// TIA Portal V15.1 export
// export: Created 2024-05-17T05:38:41.5679982Z, ExportSetting WithDefaults, DisplayName Totally Integrated Automation Portal, DisplayVersion V15.1 Update 5, DisplayName TIA Portal Openness, DisplayVersion V15.1 Update 5, DisplayName SINAMICS Startdrive Advanced, DisplayVersion V15.1, DisplayName G130, G150, S120, S150, SINAMICS MV, S210, DisplayVersion V15.1, DisplayName G110M, G120, G120C, G120D, G120P, DisplayVersion V15.1, DisplayName STEP 7 Professional, DisplayVersion V15.1 Update 5, DisplayName STEP 7 Safety, DisplayVersion V15.1, DisplayName WinCC Professional, DisplayVersion V15.1 Update 5, DisplayName SIMATIC Visualization Architect, DisplayVersion V15.1
FUNCTION "LGBLineConvBrake-MDXPN-DFS22B-Config" : Void   // FC6713, FBD
TITLE = LCrossConv2W2S-G120PN-Config / LGBLineConvBrake-MDXPN-DFS22B-Config
{ S7_Optimized_Access := 'FALSE' }
AUTHOR : VCC
FAMILY : Config
NAME : Bit2Word
VERSION : 0.1
// =============================================================================
// Handles the LCross2W2SG120PN Config
// =============================================================================
// stored: AutoNumber false, IsIECCheckEnabled false, SetENOAutomatically False, UDAEnableTagReadback false
   VAR_INPUT
      C_DetBeltTensionUsed : Bool;   // Input 0 / Config / Lowspeed stop detection Set used
      C_DetMinGapLeftUsed : Bool;   // Input 0 / Config / Lowspeed stop detection Set used
      C_DetMinGapRightUsed : Bool;   // Input 0 / Config / Lowspeed stop detection Set used
      C_BothDetMinGapIsAlarmB : Bool;   // Config
      C_OneDetMinGapIsAlarmC : Bool;   // Config
      C_InitDirectionMotPower : Bool;   // Input 7 / Config
      C_InitDirectionMotBrake : Bool;   // Input 7 / Config
      C_SafetySwNcMotPower : Bool;   // Input 15 / Config
      C_SafetySwUsedMotPower : Bool;   // Input 16 / Config
      C_SafetySwNcMotBrake : Bool;   // Input 15 / Config
      C_SafetySwUsedMotBrake : Bool;   // Input 16 / Config
      C_MotorProtectionNc : Bool;   // Motorprotection NC / Config
      C_MotorProtectionUsed : Bool;   // Motorprotection NC / Config
      C_BrakeProtectionNc : Bool;   // Config
      C_BrakeProtectionUsed : Bool;   // Config
      C_MotionStopUsed : Bool;   // Config
      C_EnableAlarmHW : Bool;   // Enable Alarm hardware (e.g. safetyswitch, motorprotector, detections) / Enable Alarm hardware (e.g. Safetyswitch, Motorprotector, detections) / Config
      C_EnableAlarmTransfer : Bool;   // Enable Alarm transfer (e.g. Transfer in , transfer out) / Config
      C_DetSaturationDelay : Time;   // Config
      C_RampMotBrake : Time;   // Config
      C_ReferenceDriveCurrentMotBrake : Real;   // Config
      C_ReferenceMotorCurrentMotBrake : Real;   // Config
      C_ReferenceMotorRPMMotBrake : Real;   // Config
      C_RatioGearboxMotBrake : Real;   // Config
      C_DiameterMotBrake : Real;   // Config
      C_AccelerationMotBrake : Real;   // Config
      C_RampMotPower : Time;   // Config
      C_ReferenceDriveCurrentMotPower : Real;   // Config
      C_ReferenceMotorCurrentMotPower : Real;   // Config
      C_ReferenceMotorRPMMotPower : Real;   // Config
      C_RatioGearboxMotPower : Real;   // Config
      C_DiameterMotPower : Real;   // Config
      C_AccelerationMotPower : Real;   // Config
      C_TrfMaxTime : DInt;   // Max allowed transfertime (millisec) / Config
      C_AllowedResetDirection : Bool;   // Config
      C_MaxTimeResetDirection : DInt;   // Config
      C_AllowedEcoMode : Bool;   // Config
      C_TimeEcoMode : Time;   // Config
      C_HWSubInputMotPower : HW_SUBMODULE;   // I/O / Config
      C_HWSubOutputMotPower : HW_SUBMODULE;   // I/O / Config
      C_HWSubInputMotBrake : HW_SUBMODULE;   // I/O / Config
      C_HWSubOutputMotBrake : HW_SUBMODULE;   // I/O / Config
   END_VAR
   VAR_IN_OUT
      IO_Config : "LineConvBrake-MDXPNConfig";   // Config
   END_VAR
BEGIN

REGION Network 1: **** 1 - Inputs **** Move Config
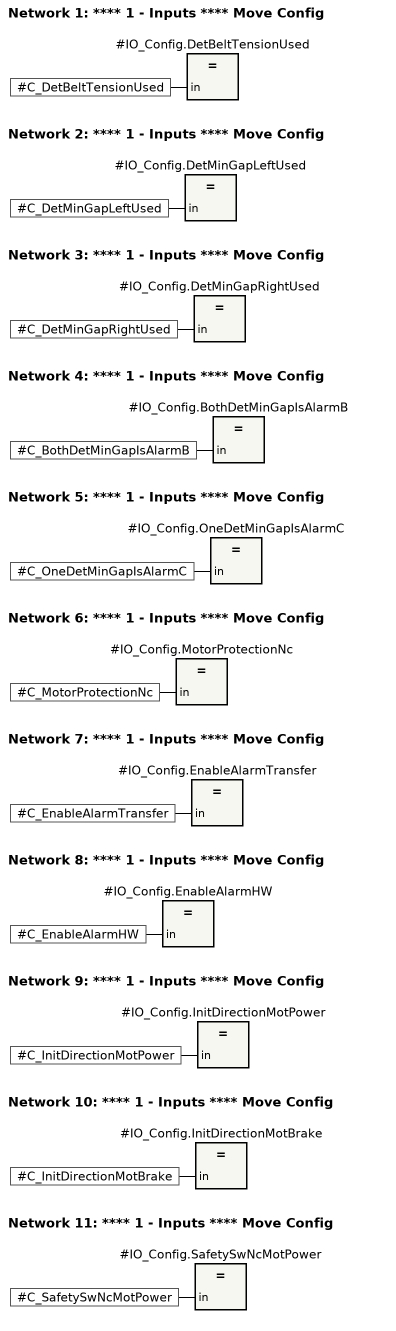
   #IO_Config.DetBeltTensionUsed := #C_DetBeltTensionUsed;
END_REGION

REGION Network 2: **** 1 - Inputs **** Move Config
   #IO_Config.DetMinGapLeftUsed := #C_DetMinGapLeftUsed;
END_REGION

REGION Network 3: **** 1 - Inputs **** Move Config
   #IO_Config.DetMinGapRightUsed := #C_DetMinGapRightUsed;
END_REGION

REGION Network 4: **** 1 - Inputs **** Move Config
   #IO_Config.BothDetMinGapIsAlarmB := #C_BothDetMinGapIsAlarmB;
END_REGION

REGION Network 5: **** 1 - Inputs **** Move Config
   #IO_Config.OneDetMinGapIsAlarmC := #C_OneDetMinGapIsAlarmC;
END_REGION

REGION Network 6: **** 1 - Inputs **** Move Config
   // Move Config
   #IO_Config.MotorProtectionNc := #C_MotorProtectionNc;
END_REGION

REGION Network 7: **** 1 - Inputs **** Move Config
   // Move Config
   #IO_Config.EnableAlarmTransfer := #C_EnableAlarmTransfer;
END_REGION

REGION Network 8: **** 1 - Inputs **** Move Config
   // Move Config
   #IO_Config.EnableAlarmHW := #C_EnableAlarmHW;
END_REGION

REGION Network 9: **** 1 - Inputs **** Move Config
   // Move Config
   #IO_Config.InitDirectionMotPower := #C_InitDirectionMotPower;
END_REGION

REGION Network 10: **** 1 - Inputs **** Move Config
   // Move Config
   #IO_Config.InitDirectionMotBrake := #C_InitDirectionMotBrake;
END_REGION

REGION Network 11: **** 1 - Inputs **** Move Config
   // Move Config
   #IO_Config.SafetySwNcMotPower := #C_SafetySwNcMotPower;
END_REGION

REGION Network 12: **** 1 - Inputs **** Move Config
   // Move Config
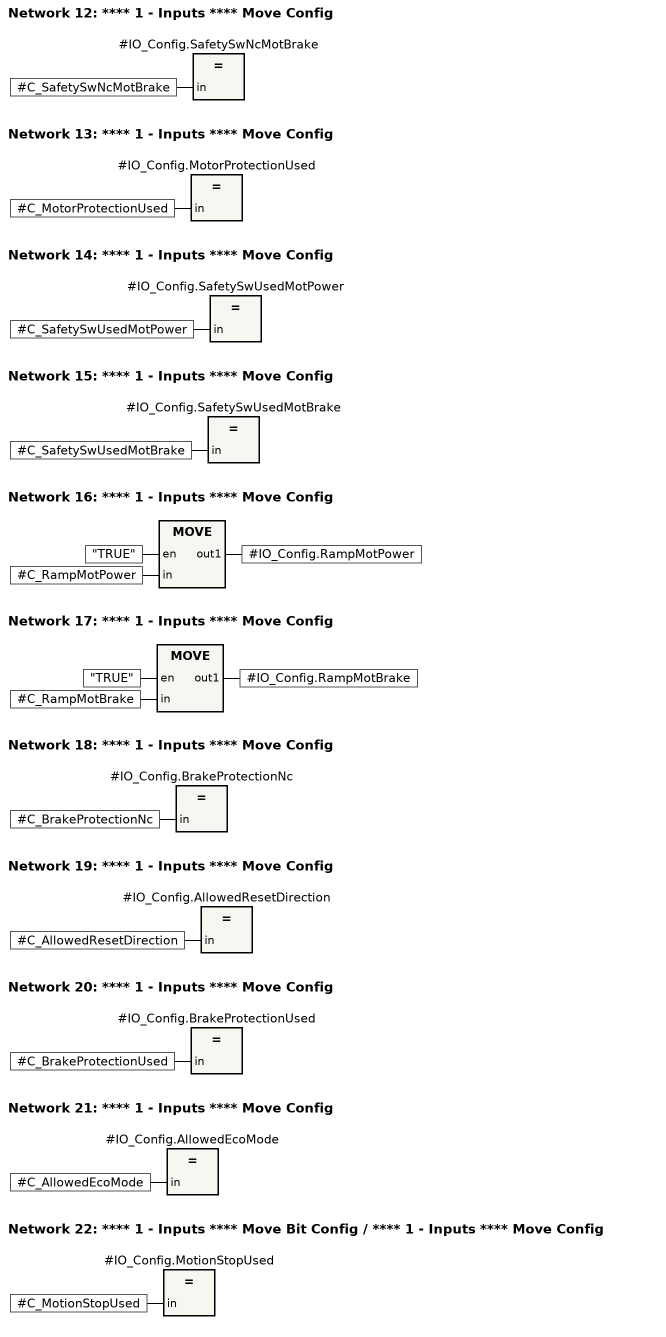
   #IO_Config.SafetySwNcMotBrake := #C_SafetySwNcMotBrake;
END_REGION

REGION Network 13: **** 1 - Inputs **** Move Config
   // Move Config
   #IO_Config.MotorProtectionUsed := #C_MotorProtectionUsed;
END_REGION

REGION Network 14: **** 1 - Inputs **** Move Config
   // Move Config
   #IO_Config.SafetySwUsedMotPower := #C_SafetySwUsedMotPower;
END_REGION

REGION Network 15: **** 1 - Inputs **** Move Config
   // Move Config
   #IO_Config.SafetySwUsedMotBrake := #C_SafetySwUsedMotBrake;
END_REGION

REGION Network 16: **** 1 - Inputs **** Move Config
   // Move Config
   IF "TRUE" THEN #IO_Config.RampMotPower := #C_RampMotPower; END_IF;
END_REGION

REGION Network 17: **** 1 - Inputs **** Move Config
   // Move Config
   IF "TRUE" THEN #IO_Config.RampMotBrake := #C_RampMotBrake; END_IF;
END_REGION

REGION Network 18: **** 1 - Inputs **** Move Config
   // Move Config
   #IO_Config.BrakeProtectionNc := #C_BrakeProtectionNc;
END_REGION

REGION Network 19: **** 1 - Inputs **** Move Config
   #IO_Config.AllowedResetDirection := #C_AllowedResetDirection;
END_REGION

REGION Network 20: **** 1 - Inputs **** Move Config
   // Move Config
   #IO_Config.BrakeProtectionUsed := #C_BrakeProtectionUsed;
END_REGION

REGION Network 21: **** 1 - Inputs **** Move Config
   // Move Config
   #IO_Config.AllowedEcoMode := #C_AllowedEcoMode;
END_REGION

REGION Network 22: **** 1 - Inputs **** Move Bit Config / **** 1 - Inputs **** Move Config
   // Move Bit Config / Move Config
   #IO_Config.MotionStopUsed := #C_MotionStopUsed;
END_REGION

NETWORK
TITLE = **** 8 - Outputs **** Move Config UDT
// Move Config
      L     #C_ReferenceMotorCurrentMotBrake;
      T     #IO_Config.ReferenceMotorCurrentMotBrake;
      L     #C_ReferenceDriveCurrentMotBrake;
      T     #IO_Config.ReferenceDriveCurrentMotBrake;
      L     #C_ReferenceMotorRPMMotBrake;
      T     #IO_Config.ReferenceMotorRPMMotBrake;
      L     #C_RatioGearboxMotBrake;
      T     #IO_Config.RatioGearboxMotBrake;
      L     #C_DiameterMotBrake;
      T     #IO_Config.DiameterMotBrake;
      L     #C_AccelerationMotBrake;
      T     #IO_Config.AccelerationMotBrake;
      L     #C_ReferenceMotorCurrentMotPower;
      T     #IO_Config.ReferenceMotorCurrentMotPower;
      L     #C_ReferenceDriveCurrentMotPower;
      T     #IO_Config.ReferenceDriveCurrentMotPower;
      L     #C_ReferenceMotorRPMMotPower;
      T     #IO_Config.ReferenceMotorRPMMotPower;
      L     #C_RatioGearboxMotPower;
      T     #IO_Config.RatioGearboxMotPower;
      L     #C_DiameterMotPower;
      T     #IO_Config.DiameterMotPower;
      L     #C_AccelerationMotPower;
      T     #IO_Config.AccelerationMotPower;


      L     #C_DetSaturationDelay;
      T     #IO_Config.DetSaturationDelay;
      L     #C_TrfMaxTime;
      T     #IO_Config.TrfMaxTime;
      L     #C_MaxTimeResetDirection;
      T     #IO_Config.MaxTimeResetDirection;
      L     #C_TimeEcoMode;
      T     #IO_Config.TimeEcoMode;
      L     #C_HWSubInputMotPower;
      T     #IO_Config.HWSubInputMotPower;
      L     #C_HWSubOutputMotPower;
      T     #IO_Config.HWSubOutputMotPower;
      L     #C_HWSubInputMotBrake;
      T     #IO_Config.HWSubInputMotBrake;
      L     #C_HWSubOutputMotBrake;
      T     #IO_Config.HWSubOutputMotBrake;

END_FUNCTION
